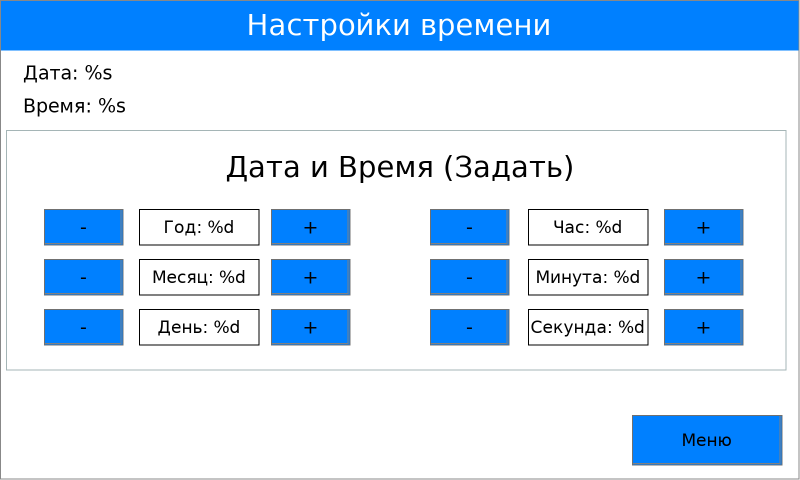
VISUALIZATION _TimeSetup_7inch  // 800x480
    RoundedRectangle (6,130 780x240)
    Rectangle (10,152 780x30), "Дата и Время (Задать)"
    RoundedRectangle (139,209 120x36), "Год: %d", text variable: TimeSetup.m_RTC.Year
        OnMouseClick: write TimeSetup.m_RTC.Set_Year via VisuDialogs.Numpad, min 1970, max 2038, title 'Year'
    RoundedRectangle (139,259 120x36), "Месяц: %d", text variable: TimeSetup.m_RTC.Month
        OnMouseClick: write TimeSetup.m_RTC.Set_Month via VisuDialogs.Numpad, min 1, max 12, title 'Month'
    RoundedRectangle (139,309 120x36), "День: %d", text variable: TimeSetup.m_RTC.Day
        OnMouseClick: write TimeSetup.m_RTC.Set_Day via VisuDialogs.Numpad, min 1, max 31, title 'Day'
    Button (44,209 79x36), "-"
        tap TimeSetup.m_RTC.Sub_Year
    Button (44,259 79x36), "-"
        tap TimeSetup.m_RTC.Sub_Month
    Button (44,309 79x36), "-"
        tap TimeSetup.m_RTC.Sub_Day
    Button (271,209 79x36), "+"
        tap TimeSetup.m_RTC.Add_Year
    Button (271,259 79x36), "+"
        tap TimeSetup.m_RTC.Add_Month
    Button (271,309 79x36), "+"
        tap TimeSetup.m_RTC.Add_Day
    RoundedRectangle (528,209 120x36), "Час: %d", text variable: TimeSetup.m_RTC.Hour
        OnMouseClick: write TimeSetup.m_RTC.Set_Hour via VisuDialogs.Numpad, min 0, max 23, title 'Hour'
    RoundedRectangle (528,259 120x36), "Минута: %d", text variable: TimeSetup.m_RTC.Minute
        OnMouseClick: write TimeSetup.m_RTC.Set_Minute via VisuDialogs.Numpad, min 0, max 59, title 'Minute'
    RoundedRectangle (528,309 120x36), "Секунда: %d", text variable: TimeSetup.m_RTC.Second
        OnMouseClick: write TimeSetup.m_RTC.Set_Second via VisuDialogs.Numpad, min 0, max 59, title 'Second'
    Button (430,209 79x36), "-"
        tap TimeSetup.m_RTC.Sub_Hour
    Button (430,259 79x36), "-"
        tap TimeSetup.m_RTC.Sub_Minute
    Button (430,309 79x36), "-"
        tap TimeSetup.m_RTC.Sub_Second
    Button (664,209 79x36), "+"
        tap TimeSetup.m_RTC.Add_Hour
    Button (664,259 79x36), "+"
        tap TimeSetup.m_RTC.Add_Minute
    Button (664,309 79x36), "+"
        tap TimeSetup.m_RTC.Add_Second
    Rectangle (20,58 400x30), "Дата: %s", text variable: TimeSetup.w_str_dateM
    Rectangle (20,91 400x30), "Время: %s", text variable: TimeSetup.w_str_time
    Button (632,415 150x50), "Меню"
        OnMouseDown:  Assign=_SettingsMain_7inch, Type=Assignment
    Rectangle (0,0 798x50), "Настройки времени"
END_VISUALIZATION

// Device/Application/Vizualization/7_inch/_Diag_supKey
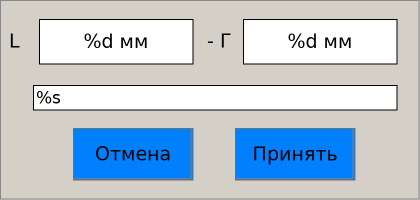
VISUALIZATION _Diag_supKey  // 420x200
VAR_IN_OUT
	stValue: SupportType2;	
END_VAR
VAR

END_VAR
    Button (235,128 120x52), "Принять"
        OnMouseDown:  Dialog=Current Dialog, Result=OK, NumpadKeypadSet=True
    Button (73,128 120x52), "Отмена"
        OnMouseClick:  Dialog=Current Dialog, Result=Cancel, NumpadKeypadSet=True
    RoundedRectangle (33,85 364x25), "%s", text variable: stValue.name
    Label (6,26 31x30), "L"
    RoundedRectangle (39,19 154x45), "%d мм", text variable: stValue.arLength[0]
        OnMouseClick: write the text variable via VisuDialogs.Numpad, min -999, max 999, title 'Input'
        OnDialogClosed: execute { stValue.name:= WCONCAT( WCONCAT("L", int_to_wstring(stValue.arLength[0])), WCONCAT(" - Г", int_to_wstring(stValue.arLength[1])) ); }
    RoundedRectangle (243,19 154x45), "%d мм", text variable: stValue.arLength[1]
        OnMouseClick: write the text variable via VisuDialogs.Numpad, min -999, max 999, title 'Input'
        OnDialogClosed: execute { stValue.name:= WCONCAT( WCONCAT("L", int_to_wstring(stValue.arLength[0])), WCONCAT(" - Г", int_to_wstring(stValue.arLength[1])) ); }
    Label (204,26 31x30), "- Г"
END_VISUALIZATION

(* text list OnOffList (id | default)
  0 | Выкл.
  1 | Вкл.
   |  *)

(* text list MbBoud (id | default)
  0 | 4800
  1 | 9600
  2 | 19200
  3 | 38400
  4 | 57600
  5 | 115200
   |  *)

(* text list NoYes (id | default)
  0 | Нет
  1 | Да
   |  *)

(* text list ModeSysList (id | default)
  0 | Режим: Цикличный
  1 | Режим: Прерывистый
  2 | Режим: Ручной
   |  *)

(* text list typeEquip (id | default)
  0 | N
  1 | F
   |  *)

(* text list Direction (id | default)
  0 | L
  1 | R
   |  *)

(* text list AlarmGroup (id | default)
  9 | Ошибка драйвера актуатора 2
  8 | Ошибка драйвера актуатора 1
  7 | Нет сигнала с модулем ПР
  6 | Достигнута минимально крайняя точка движения (координата X3)
  5 | Достигнута максимально крайняя точка движения (координата X4)
  4 | Проведите плановое плановое ТО
  3 | Ошибка дижения рабочего цилиндра
  2 | Ошибка датчика линейного перемещения
  1 | Сработало тепловое реле элекродвигателя маслостанции
  0 | Нажата кнопка аварийного останова
   |  *)

(* text list MbParity (id | default)
  2 | Чет
  0 | Нет
  1 | Нечет
   |  *)

(* text list MbStopbit (id | default)
  1 | 1
  2 | 2
  3 | 1.5
   |  *)

(* text list WarningGroup (id | default)
  2 | Нет подходящей поддержки
  1 | Расчитанных ход актуаторов больше, чем их возможный
  0 | Начальная позиция актуаторов выходит за допустимы предел
   |  *)

(* text list TypeSetup (id | default)
  0 | L
  1 | Г
   |  *)

(* text list DirectRotation (id | default)
  0 | Правое
  1 | Левое
   |  *)
